// instrument joints control
FUNCTION_BLOCK FB_UltrosonicKnifeControl_old
VAR_INPUT
END_VAR
VAR_OUTPUT
END_VAR
VAR
	// instrument PID control paramters
	m_instruKp:ARRAY[1..5] OF LREAL:=[5(5)];
	m_instruKd:ARRAY[1..5] OF LREAL:=[5(0.25)];
	m_instruKi:ARRAY[1..5] OF LREAL:=[5(10.0)];
	m_instruKiLimit:ARRAY[1..5] OF LREAL:=[5(100.0)];
	m_instruCtrlLimit:ARRAY[1..5] OF LREAL:=[3(200.0), 2(350.0)];
	
	// max grip force/current(mA)
	m_maxGripForce:LREAL;
	m_maxGripCurrent:LREAL:=200.0;
	
	// PID for instrument joint position
	m_instruJntCtrl:ARRAY[1..5] OF FB_PID;

	// command instrument joint position and velocity
	m_instruCmdJntPos:Vec5d;
	m_instruLastCmdJntPos:Vec5d;
	m_instruCmdJntVel:Vec5d;
	
	// backlash compensation variables
	m_jntBacklash:ARRAY[1..5] OF LREAL:=[5(0)];
	m_jntMoveStep:LREAL := 0.5*g_deg2Rad;
	
	// current instrument joint position and velocity
	m_instruCurJntPos: Vec5d;
	m_instruCurJntVel:Vec5d;
	
	// grasp force level
	m_graspForceLevel:Lreal :=0;
	
	// instrument joint control torque(when gripper is open)
	m_instruJntCtrlTrq:Vec5d:=[5(0.0)];
	
	// minimum grip angle to apply grip force; convert grasp force level to minus grip angle
	m_minGripAngle :LREAL := -60*g_deg2Rad;
	m_gripForceAngle:LREAL;
	
END_VAR

METHOD calcBacklash : BOOL
VAR_IN_OUT CONSTANT
	// instrument joint command position
	i_cmdInstruJntPos :Vec5d;
	
	// slave arm data
	i_slaveArm :FB_SlaveArm;
END_VAR

VAR
	i:INT;
	deltaAng:LREAL;
END_VAR
// backslash compensation
FOR i:=3 TO 3 DO
	// integral compensated backslash angle
	deltaAng:=i_cmdInstruJntPos[i]-m_instruLastCmdJntPos[i];
	IF ABS(deltaAng)>m_jntMoveStep THEN
		m_jntBacklash [i] := m_jntBacklash [i] + m_jntMoveStep*sign(deltaAng);
		m_instruLastCmdJntPos[i] := i_cmdInstruJntPos[i];
	END_IF
END_FOR


// exert grip force 
IF m_graspForceLevel >0  THEN
	
	// max grip finger backlash
	m_jntBacklash [3]:=-i_slaveArm.instrument.instruTypeInfo.m_instruYawBacklash;
	
END_IF

// limit compensated backslash angle
FOR i:=3 TO 3 DO
	IF g_instruBacklashDir[i] > 0 THEN
		m_jntBacklash [i] := LIMIT(0, m_jntBacklash[i], i_slaveArm.instrument.instruTypeInfo.m_instruYawBacklash);
	ELSE
		m_jntBacklash [i] := LIMIT(-i_slaveArm.instrument.instruTypeInfo.m_instruYawBacklash, m_jntBacklash[i], 0);	
	END_IF
	
END_FOR
END_METHOD

METHOD init : BOOL
VAR_IN_OUT CONSTANT
	i_slaveArm:FB_SlaveArm;
END_VAR

VAR
	i,j:INT;
	currentRatioMotor2Jnt:LREAL;
END_VAR
m_graspForceLevel:=0;

// init controller
currentRatioMotor2Jnt:=GVL_SlaveMotorParameters.g_motorTrqConst[4]*GVL_SlaveMotorParameters.g_motorReduction[4]/1000;
m_maxGripForce := m_maxGripCurrent * currentRatioMotor2Jnt;
FOR i:=1 TO 5 DO
	m_jntBacklash[i] := 0;
	m_instruCmdJntPos[i]:=i_slaveArm.curJntPos[i+3];
	m_instruLastCmdJntPos[i]:=m_instruCmdJntPos[i];
	m_instruCmdJntVel[i]:=0;
	
	m_instruJntCtrl[i].init(g_slaveArmCtrlCycleTime,m_instruKp[i],m_instruKd[i],m_instruKi[i],
		m_instruKiLimit[i]* currentRatioMotor2Jnt,	m_instruCtrlLimit[i]*currentRatioMotor2Jnt);
END_FOR
END_METHOD

METHOD run : BOOL
VAR_IN_OUT CONSTANT
	// instrument joint command position
	i_cmdInstruJntPos :Vec5d;
	
	// instrument joint command velocity
	i_cmdInstruJntVel :Vec5d;
	
	// command grip force level
	i_cmdGripForceLevel:LREAL;
	
	// slave arm data
	i_slaveArm :FB_SlaveArm;
END_VAR

VAR_OUTPUT
	// joint control torque
	o_cmdJntTrq:Vec5d;
END_VAR

VAR
	i: INT;
END_VAR
// calculate instrument backlash
calcBacklash(i_cmdInstruJntPos, i_slaveArm);

// convert force level to grip angle
m_graspForceLevel:=LIMIT(0,i_cmdGripForceLevel , 100);
m_gripForceAngle:=m_minGripAngle*m_graspForceLevel/100;

// joint position control
FOR i:=1 TO 5 DO	
	m_instruCmdJntPos[i]:=i_cmdInstruJntPos[i];
	m_instruCmdJntVel[i]:=i_cmdInstruJntVel[i];
	m_instruCurJntPos[i]:=i_slaveArm.curJntPos[i+3];
	m_instruCurJntVel[i]:= i_slaveArm.curJntVel[i+3];
	IF i=3 THEN
		m_instruCmdJntPos[i]:=i_cmdInstruJntPos[i]+m_gripForceAngle;
	END_IF
	m_instruJntCtrlTrq[i]:=m_instruJntCtrl[i].run(m_instruCmdJntPos[i]+ m_jntBacklash[i] ,m_instruCurJntPos[i], m_instruCmdJntVel[i], m_instruCurJntVel[i]);
END_FOR
m_instruJntCtrlTrq[1]:=0;
m_instruJntCtrlTrq[2]:=0;
m_instruJntCtrlTrq[4]:=0.5*m_instruJntCtrlTrq[5];

// exert grip force 
//IF m_graspForceLevel >0  THEN
//	m_instruJntCtrlTrq[3]:= -m_maxGripForce*m_graspForceLevel/100.0;	
//END_IF

o_cmdJntTrq := m_instruJntCtrlTrq;
END_METHOD

END_FUNCTION_BLOCK

(* stored: Version 1.1.0.1, ProductVersion 3.1.4024.11
   POU FB_UltrosonicKnifeControl_old: Id {675f3909-c472-4838-a346-da9f4950f3d4}, SpecialFunc None
   Method calcBacklash: Id {aab45778-dc4d-45b7-982f-1304e391e20f}
   Method init: Id {6e920412-a4cf-4cf4-9a5a-71c3a35e14a6}
   Method run: Id {21647c6f-a530-4d8b-818e-e8fe9b57826d} *)
